PROGRAM INIT

VAR
	once: BOOL := FALSE;
END_VAR

IF(once=FALSE)THEN
	ENC.DEG_TO_INC := UDINT_TO_DINT(SDO.enc_resolution/360);
	ENC.RPM_TO_INCS:= UDINT_TO_DINT(SDO.enc_resolution/60);
	MOTOR.GEAR_RATIO := UDINT_TO_DINT(SDO.motor_revolutions/SDO.shaft_revolutions);
	MOTOR.RATED_TORQUE_NM 	:= DINT_TO_LREAL(SDO.motor_rated_torque)/1000.0;	
	MOTOR.RATED_SPEED_RPM	:= SDO.max_motor_speed/1000;
	once := TRUE;
END_IF

END_PROGRAM

(* stored: Version 1.1.0.1, ProductVersion 3.1.4024.11
   POU INIT: Id {fe257ffe-7e53-4cf4-b90e-41c71454b463}, SpecialFunc None *)
